Staubli VAL3: sendRosMsg.pgx

public program sendRosMsg(sio& x_sTcpSocket, Prefix& x_pPrefix, Header& x_hHeader, Body& x_bBody, num& x_nConnFlag)
begin
  // Copyright (c) 2016, Ocado Technology - Robotics Research Team
  //
  // Licensed under the Apache License, Version 2.0 (the "License");
  // you may not use this file except in compliance with the License.
  // You may obtain a copy of the License at
  //
  //     http://www.apache.org/licenses/LICENSE-2.0
  //
  // Unless required by applicable law or agreed to in writing, software
  // distributed under the License is distributed on an "AS IS" BASIS,
  // WITHOUT WARRANTIES OR CONDITIONS OF ANY KIND, either express or implied.
  // See the License for the specific language governing permissions and
  // limitations under the License.



  call sendData(x_sTcpSocket, x_pPrefix.nData, x_nConnFlag)
  call sendData(x_sTcpSocket, x_hHeader.nData, x_nConnFlag)
  call sendData(x_sTcpSocket, x_bBody.nData, x_nConnFlag)
end
